PROGRAM MAIN
VAR
END_VAR

END_PROGRAM

(* stored: Version 1.1.0.1
   POU MAIN: Id {72c2ee86-1d0b-498b-a1ff-b3a7280d4623} *)
